// TIA Portal V20 export
TYPE "LER_typeLaserMarkTrackingData"
// stored: Access Published
   STRUCT
      resultData { ExternalWritable := 'False'} : String[32];
      ngDataComplete { ExternalWritable := 'False'} : Bool;
      okDataComplete { ExternalWritable := 'False'} : Bool;
   END_STRUCT;
END_TYPE
